TYPE ScriblyComSubscribe :
STRUCT
  Request : ScriblyComRequest; // contains booleans that are used to start a specific sequence.
  Equipment : ScriblyComSubscribeEquipment;  // structs for equipment objects which are used by the bridges
  
  Segments : ScriblyComSubscribeSegments;
END_STRUCT
END_TYPE

(* stored: Version 1.1.0.1
   DUT ScriblyComSubscribe: Id {4e2bd3b8-056c-42c7-908e-5d1fd01b59e7} *)
